FUNCTION_BLOCK LevelDifferenceSD (* Basic Function Block Type *)
  (* Standard: 61499-2 *)
  (* Version 0.0, 7/13/2026, Schneider Electric, Template *)
  PACKAGE SE.Nereda;
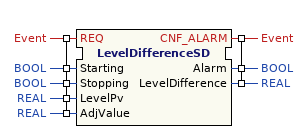
  EVENT_INPUT
    REQ WITH Starting, Stopping, LevelPv, AdjValue; (* Normal Execution Request *)
  END_EVENT
  EVENT_OUTPUT
    CNF_ALARM WITH Alarm, LevelDifference; (* Execution Confirmation *)
  END_EVENT
  VAR_INPUT
    Starting : BOOL;
    Stopping : BOOL;
    LevelPv : REAL;
    AdjValue : REAL;
  END_VAR
  VAR_OUTPUT
    Alarm : BOOL;
    LevelDifference : REAL;
  END_VAR
  VAR
    MemoLevelPv : REAL;
    LevelDiff : REAL;
  END_VAR
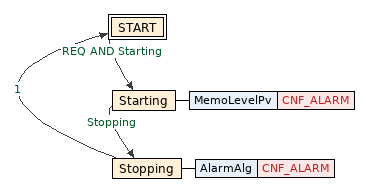
  EC_STATES
    START; (* Initial State *)
    Starting : MemoLevelPv -> CNF_ALARM;
    Stopping : AlarmAlg -> CNF_ALARM;
  END_STATES
  EC_TRANSITIONS
    START TO Starting := REQ AND Starting;
    Stopping TO START := 1;
    Starting TO Stopping := Stopping;
  END_TRANSITIONS
  ALGORITHM MemoLevelPv IN ST:
;
MemoLevelPv := LevelPv;
Alarm := FALSE;
  END_ALGORITHM
  ALGORITHM AlarmAlg IN ST:
;
LevelDiff := MemoLevelPv - LevelPv;
LevelDifference := MemoLevelPv - LevelPv;

IF LevelDiff < AdjValue THEN
	Alarm := TRUE;
ELSE
	Alarm := FALSE;
END_IF;
  END_ALGORITHM
END_FUNCTION_BLOCK
